PROGRAM BH0IPL_LineBackground
VAR
END_VAR

MAIN.stLine_BH0IPL.fbLine(stLine:=MAIN.stLine_BH0IPL);
MAIN.stLine_BH0IPL.stStation_BH0IPL01.fbStation(
				stLine:=MAIN.stLine_BH0IPL,
				stStation:=MAIN.stLine_BH0IPL.stStation_BH0IPL01);

END_PROGRAM

(* stored: Version 1.1.0.1, ProductVersion 3.1.4024.15
   POU BH0IPL_LineBackground: Id {5458bbde-d293-423e-a9c5-117cf7db0055}, SpecialFunc None *)
